	fbSetExtendedFadeTime.ipDALICommunication := ipDALICommunication;
	fbSetFadeRate.ipDALICommunication := ipDALICommunication;
	fbSetFadeTime.ipDALICommunication := ipDALICommunication;
{endregion}
10:
{region "Query Fade Time and Fade Rate"}
	fbQueryFadeTimeFadeRate(bStart := TRUE,
							nAddress := nAddress,
							eAddressType := eAddressType,
							eCommandPriority := E_DALICommandPriority.Middle,
							eFadeTime=> eFadeTime,
							eFadeRate=> eFadeRate);
	IF (NOT fbQueryFadeTimeFadeRate.bBusy) THEN
		fbQueryFadeTimeFadeRate(bStart := FALSE);
		IF (eFadeTime = 0) THEN 
			bNoFadeTime := FALSE; // Check whether Fade Time is available
			nStep := 20;
		ELSE 	 
			bNoFadeTime := TRUE;
			nStep := 0;
		END_IF
	END_IF
{endregion}
20:
{region "Query Extended Fade Time"}
	fbQueryExtendedFadeTime(bStart := TRUE,
							nAddress := nAddress,
							eAddressType := eAddressType,
							eCommandPriority := E_DALICommandPriority.Middle,
							eExtendedFadeTimeBase=> eExtendedFadeTimeBase,
							eExtendedFadeTimeMultiplier=> eExtendedFadeTimeMultiplier);
	IF (NOT fbQueryExtendedFadeTime.bBusy) THEN
		fbQueryExtendedFadeTime(bStart := FALSE);
		nStep := 0;
		IF (eExtendedFadeTimeMultiplier = E_DALIExtendedFadeTimeMultiplier.Disabled) THEN
			eExtendedFadeTime := E_DALIExtendedFadeTime.NoFade;
		END_IF
		IF (eExtendedFadeTimeMultiplier = E_DALIExtendedFadeTimeMultiplier.Multiplier100ms) THEN
			CASE eExtendedFadeTimeBase OF
				E_DALIExtendedFadeTimeBase.Base01:	eExtendedFadeTime := E_DALIExtendedFadeTime.onehundred;
				E_DALIExtendedFadeTimeBase.Base02:	eExtendedFadeTime := E_DALIExtendedFadeTime.twohundred;
				E_DALIExtendedFadeTimeBase.Base03:	eExtendedFadeTime := E_DALIExtendedFadeTime.threehundred;
				E_DALIExtendedFadeTimeBase.Base04:	eExtendedFadeTime := E_DALIExtendedFadeTime.fourhundred;
				E_DALIExtendedFadeTimeBase.Base05:	eExtendedFadeTime := E_DALIExtendedFadeTime.fivehundred;
				E_DALIExtendedFadeTimeBase.Base06:	eExtendedFadeTime := E_DALIExtendedFadeTime.sixhundred;
				E_DALIExtendedFadeTimeBase.Base07:	eExtendedFadeTime := E_DALIExtendedFadeTime.sevenhundred;
				E_DALIExtendedFadeTimeBase.Base08:	eExtendedFadeTime := E_DALIExtendedFadeTime.eighthundred;
				E_DALIExtendedFadeTimeBase.Base09:	eExtendedFadeTime := E_DALIExtendedFadeTime.ninehundred;
				E_DALIExtendedFadeTimeBase.Base10:	eExtendedFadeTime := E_DALIExtendedFadeTime.onethousand;
				E_DALIExtendedFadeTimeBase.Base11:	eExtendedFadeTime := E_DALIExtendedFadeTime.onethousandonehundred;
				E_DALIExtendedFadeTimeBase.Base12:	eExtendedFadeTime := E_DALIExtendedFadeTime.onethousandtwohundred;
				E_DALIExtendedFadeTimeBase.Base13:	eExtendedFadeTime := E_DALIExtendedFadeTime.onethousandthreehundred;
				E_DALIExtendedFadeTimeBase.Base14:	eExtendedFadeTime := E_DALIExtendedFadeTime.onethousandfourhundred;
				E_DALIExtendedFadeTimeBase.Base15:	eExtendedFadeTime := E_DALIExtendedFadeTime.onethousandfivehundred;
				E_DALIExtendedFadeTimeBase.Base16:	eExtendedFadeTime := E_DALIExtendedFadeTime.onethousandsixhundred;
			END_CASE
		END_IF
	 	IF (eExtendedFadeTimeMultiplier = E_DALIExtendedFadeTimeMultiplier.Multiplier1s) THEN
			CASE eExtendedFadeTimeBase OF
				E_DALIExtendedFadeTimeBase.Base01:	eExtendedFadeTime := E_DALIExtendedFadeTime.onesecond;
				E_DALIExtendedFadeTimeBase.Base02:	eExtendedFadeTime := E_DALIExtendedFadeTime.twoseconds;
				E_DALIExtendedFadeTimeBase.Base03:	eExtendedFadeTime := E_DALIExtendedFadeTime.threeseconds;
				E_DALIExtendedFadeTimeBase.Base04:	eExtendedFadeTime := E_DALIExtendedFadeTime.fourseconds;
				E_DALIExtendedFadeTimeBase.Base05:	eExtendedFadeTime := E_DALIExtendedFadeTime.fiveseconds;
				E_DALIExtendedFadeTimeBase.Base06:	eExtendedFadeTime := E_DALIExtendedFadeTime.sixseconds;
				E_DALIExtendedFadeTimeBase.Base07:	eExtendedFadeTime := E_DALIExtendedFadeTime.sevenseconds;
				E_DALIExtendedFadeTimeBase.Base08:	eExtendedFadeTime := E_DALIExtendedFadeTime.eightseconds;
				E_DALIExtendedFadeTimeBase.Base09:	eExtendedFadeTime := E_DALIExtendedFadeTime.nineseconds;
				E_DALIExtendedFadeTimeBase.Base10:	eExtendedFadeTime := E_DALIExtendedFadeTime.tenseconds;
				E_DALIExtendedFadeTimeBase.Base11:	eExtendedFadeTime := E_DALIExtendedFadeTime.elevenseconds;
				E_DALIExtendedFadeTimeBase.Base12:	eExtendedFadeTime := E_DALIExtendedFadeTime.twelveseconds;
				E_DALIExtendedFadeTimeBase.Base13:	eExtendedFadeTime := E_DALIExtendedFadeTime.thirteenseconds;
				E_DALIExtendedFadeTimeBase.Base14:	eExtendedFadeTime := E_DALIExtendedFadeTime.fourteenseconds;
				E_DALIExtendedFadeTimeBase.Base15:	eExtendedFadeTime := E_DALIExtendedFadeTime.fifteenseconds;
				E_DALIExtendedFadeTimeBase.Base16:	eExtendedFadeTime := E_DALIExtendedFadeTime.sixteenseconds;
			END_CASE
		END_IF
		IF (eExtendedFadeTimeMultiplier = E_DALIExtendedFadeTimeMultiplier.Multiplier10s) THEN
			CASE eExtendedFadeTimeBase OF
				E_DALIExtendedFadeTimeBase.Base01:	eExtendedFadeTime := E_DALIExtendedFadeTime.ten1seconds;
				E_DALIExtendedFadeTimeBase.Base02:	eExtendedFadeTime := E_DALIExtendedFadeTime.twentyseconds;
				E_DALIExtendedFadeTimeBase.Base03:	eExtendedFadeTime := E_DALIExtendedFadeTime.thirtyseconds;
				E_DALIExtendedFadeTimeBase.Base04:	eExtendedFadeTime := E_DALIExtendedFadeTime.fourtyseconds;
				E_DALIExtendedFadeTimeBase.Base05:	eExtendedFadeTime := E_DALIExtendedFadeTime.fiftyseconds;
				E_DALIExtendedFadeTimeBase.Base06:	eExtendedFadeTime := E_DALIExtendedFadeTime.sixtyseconds;
				E_DALIExtendedFadeTimeBase.Base07:	eExtendedFadeTime := E_DALIExtendedFadeTime.seventyseconds;
				E_DALIExtendedFadeTimeBase.Base08:	eExtendedFadeTime := E_DALIExtendedFadeTime.eightyseconds;
				E_DALIExtendedFadeTimeBase.Base09:	eExtendedFadeTime := E_DALIExtendedFadeTime.ninetyseconds;
				E_DALIExtendedFadeTimeBase.Base10:	eExtendedFadeTime := E_DALIExtendedFadeTime.onehundredseconds;
				E_DALIExtendedFadeTimeBase.Base11:	eExtendedFadeTime := E_DALIExtendedFadeTime.onehundredtenseconds;
				E_DALIExtendedFadeTimeBase.Base12:	eExtendedFadeTime := E_DALIExtendedFadeTime.onehundredtwentyseconds;
				E_DALIExtendedFadeTimeBase.Base13:	eExtendedFadeTime := E_DALIExtendedFadeTime.onehundredthirtyseconds;
				E_DALIExtendedFadeTimeBase.Base14:	eExtendedFadeTime := E_DALIExtendedFadeTime.onehundredfourtyseconds;
				E_DALIExtendedFadeTimeBase.Base15:	eExtendedFadeTime := E_DALIExtendedFadeTime.onehundredfiftyseconds;
				E_DALIExtendedFadeTimeBase.Base16:	eExtendedFadeTime := E_DALIExtendedFadeTime.onehundredsixtyseconds;
			END_CASE
		END_IF
		IF (eExtendedFadeTimeMultiplier = E_DALIExtendedFadeTimeMultiplier.Multiplier1min) THEN
			CASE eExtendedFadeTimeBase OF
				E_DALIExtendedFadeTimeBase.Base01:	eExtendedFadeTime := E_DALIExtendedFadeTime.oneminute;
				E_DALIExtendedFadeTimeBase.Base02:	eExtendedFadeTime := E_DALIExtendedFadeTime.twominutes;
				E_DALIExtendedFadeTimeBase.Base03:	eExtendedFadeTime := E_DALIExtendedFadeTime.threeminutes;
				E_DALIExtendedFadeTimeBase.Base04:	eExtendedFadeTime := E_DALIExtendedFadeTime.fourminutes;
				E_DALIExtendedFadeTimeBase.Base05:	eExtendedFadeTime := E_DALIExtendedFadeTime.fiveminutes;
				E_DALIExtendedFadeTimeBase.Base06:	eExtendedFadeTime := E_DALIExtendedFadeTime.sixminutes;
				E_DALIExtendedFadeTimeBase.Base07:	eExtendedFadeTime := E_DALIExtendedFadeTime.sevenminutes;
				E_DALIExtendedFadeTimeBase.Base08:	eExtendedFadeTime := E_DALIExtendedFadeTime.eightminutes;
				E_DALIExtendedFadeTimeBase.Base09:	eExtendedFadeTime := E_DALIExtendedFadeTime.nineminutes;
				E_DALIExtendedFadeTimeBase.Base10:	eExtendedFadeTime := E_DALIExtendedFadeTime.tenminutes;
				E_DALIExtendedFadeTimeBase.Base11:	eExtendedFadeTime := E_DALIExtendedFadeTime.elevenminutes;
				E_DALIExtendedFadeTimeBase.Base12:	eExtendedFadeTime := E_DALIExtendedFadeTime.twelveminutes;
				E_DALIExtendedFadeTimeBase.Base13:	eExtendedFadeTime := E_DALIExtendedFadeTime.thirteenminutes;
				E_DALIExtendedFadeTimeBase.Base14:	eExtendedFadeTime := E_DALIExtendedFadeTime.fourteenminutes;
				E_DALIExtendedFadeTimeBase.Base15:	eExtendedFadeTime := E_DALIExtendedFadeTime.fifteenminutes;
				E_DALIExtendedFadeTimeBase.Base16:	eExtendedFadeTime := E_DALIExtendedFadeTime.sixteenminutes;
			END_CASE
		END_IF
	ELSE
		eExtendedFadeTime := E_DALIExtendedFadeTime.unknown;
	END_IF
{endregion}
1000:
{region "Set Fade Time"}
	fbSetFadeTime(bStart:= TRUE,
				  nAddress:= nAddress,
				  eAddressType := eAddressType,
				  eCommandPriority := E_DALICommandPriority.Middle,
				  eFadeTime := eFadeTime);
	IF (NOT fbSetFadeTime.bBusy) THEN
		fbSetFadeTime(bStart := FALSE);
		{region " Display whether Fade Time is available²}
		IF (eFadeTime = 0) THEN
			bNoFadeTime := FALSE;
		ELSE
			bNoFadeTime := TRUE;
		END_IF
		{endregion}
		nStep := 0;
	END_IF
{endregion}
1010:
{region "Set Fade Rate"}
	fbSetFadeRate(bStart:= TRUE,
				  nAddress:= nAddress,
				  eAddressType := eAddressType,
				  eCommandPriority := E_DALICommandPriority.Middle,
				  eFadeRate := eFadeRate);
	IF (NOT fbSetFadeRate.bBusy) THEN
		fbSetFadeRate(bStart := FALSE);
		nStep := 0;
	END_IF
{endregion}
1020:
{region "Set Extended Fade Time"}
	CASE eExtendedFadeTime OF
		E_DALIExtendedFadeTime.NoFade:					eExtendedFadeTimeBase := E_DALIExtendedFadeTimeBase.Unknown;
														eExtendedFadeTimeMultiplier := E_DALIExtendedFadeTimeMultiplier.Disabled;
		E_DALIExtendedFadeTime.onehundred:				eExtendedFadeTimeBase := E_DALIExtendedFadeTimeBase.Base01;
														eExtendedFadeTimeMultiplier := E_DALIExtendedFadeTimeMultiplier.Multiplier100ms;
		E_DALIExtendedFadeTime.twohundred:				eExtendedFadeTimeBase := E_DALIExtendedFadeTimeBase.Base02;
														eExtendedFadeTimeMultiplier := E_DALIExtendedFadeTimeMultiplier.Multiplier100ms;
		E_DALIExtendedFadeTime.threehundred:			eExtendedFadeTimeBase := E_DALIExtendedFadeTimeBase.Base03;
														eExtendedFadeTimeMultiplier := E_DALIExtendedFadeTimeMultiplier.Multiplier100ms;
		E_DALIExtendedFadeTime.fourhundred:				eExtendedFadeTimeBase := E_DALIExtendedFadeTimeBase.Base04;
														eExtendedFadeTimeMultiplier := E_DALIExtendedFadeTimeMultiplier.Multiplier100ms;
		E_DALIExtendedFadeTime.fivehundred:				eExtendedFadeTimeBase := E_DALIExtendedFadeTimeBase.Base05;
														eExtendedFadeTimeMultiplier := E_DALIExtendedFadeTimeMultiplier.Multiplier100ms;
		E_DALIExtendedFadeTime.sixhundred:				eExtendedFadeTimeBase := E_DALIExtendedFadeTimeBase.Base06;
														eExtendedFadeTimeMultiplier := E_DALIExtendedFadeTimeMultiplier.Multiplier100ms;
		E_DALIExtendedFadeTime.sevenhundred:			eExtendedFadeTimeBase := E_DALIExtendedFadeTimeBase.Base07;
														eExtendedFadeTimeMultiplier := E_DALIExtendedFadeTimeMultiplier.Multiplier100ms;
		E_DALIExtendedFadeTime.eighthundred:			eExtendedFadeTimeBase := E_DALIExtendedFadeTimeBase.Base08;
														eExtendedFadeTimeMultiplier := E_DALIExtendedFadeTimeMultiplier.Multiplier100ms;
		E_DALIExtendedFadeTime.ninehundred:				eExtendedFadeTimeBase := E_DALIExtendedFadeTimeBase.Base09;
														eExtendedFadeTimeMultiplier := E_DALIExtendedFadeTimeMultiplier.Multiplier100ms;
		E_DALIExtendedFadeTime.onethousand:				eExtendedFadeTimeBase := E_DALIExtendedFadeTimeBase.Base10;
														eExtendedFadeTimeMultiplier := E_DALIExtendedFadeTimeMultiplier.Multiplier100ms;
		E_DALIExtendedFadeTime.onethousandonehundred:	eExtendedFadeTimeBase := E_DALIExtendedFadeTimeBase.Base11;
														eExtendedFadeTimeMultiplier := E_DALIExtendedFadeTimeMultiplier.Multiplier100ms;
		E_DALIExtendedFadeTime.onethousandtwohundred:	eExtendedFadeTimeBase := E_DALIExtendedFadeTimeBase.Base12;
														eExtendedFadeTimeMultiplier := E_DALIExtendedFadeTimeMultiplier.Multiplier100ms;
		E_DALIExtendedFadeTime.onethousandthreehundred:	eExtendedFadeTimeBase := E_DALIExtendedFadeTimeBase.Base13;
														eExtendedFadeTimeMultiplier := E_DALIExtendedFadeTimeMultiplier.Multiplier100ms;
		E_DALIExtendedFadeTime.onethousandfourhundred:	eExtendedFadeTimeBase := E_DALIExtendedFadeTimeBase.Base14;
														eExtendedFadeTimeMultiplier := E_DALIExtendedFadeTimeMultiplier.Multiplier100ms;
		E_DALIExtendedFadeTime.onethousandfivehundred:	eExtendedFadeTimeBase := E_DALIExtendedFadeTimeBase.Base15;
														eExtendedFadeTimeMultiplier := E_DALIExtendedFadeTimeMultiplier.Multiplier100ms;
		E_DALIExtendedFadeTime.onethousandsixhundred:	eExtendedFadeTimeBase := E_DALIExtendedFadeTimeBase.Base16;
														eExtendedFadeTimeMultiplier := E_DALIExtendedFadeTimeMultiplier.Multiplier100ms;
		E_DALIExtendedFadeTime.onesecond:				eExtendedFadeTimeBase := E_DALIExtendedFadeTimeBase.Base01;
														eExtendedFadeTimeMultiplier := E_DALIExtendedFadeTimeMultiplier.Multiplier1s;
		E_DALIExtendedFadeTime.twoseconds:				eExtendedFadeTimeBase := E_DALIExtendedFadeTimeBase.Base02;
														eExtendedFadeTimeMultiplier := E_DALIExtendedFadeTimeMultiplier.Multiplier1s;
		E_DALIExtendedFadeTime.threeseconds:			eExtendedFadeTimeBase := E_DALIExtendedFadeTimeBase.Base03;
														eExtendedFadeTimeMultiplier := E_DALIExtendedFadeTimeMultiplier.Multiplier1s;
		E_DALIExtendedFadeTime.fourseconds:				eExtendedFadeTimeBase := E_DALIExtendedFadeTimeBase.Base04;
														eExtendedFadeTimeMultiplier := E_DALIExtendedFadeTimeMultiplier.Multiplier1s;
		E_DALIExtendedFadeTime.fiveseconds:				eExtendedFadeTimeBase := E_DALIExtendedFadeTimeBase.Base05;
														eExtendedFadeTimeMultiplier := E_DALIExtendedFadeTimeMultiplier.Multiplier1s;
		E_DALIExtendedFadeTime.sixseconds:				eExtendedFadeTimeBase := E_DALIExtendedFadeTimeBase.Base06;
														eExtendedFadeTimeMultiplier := E_DALIExtendedFadeTimeMultiplier.Multiplier1s;
		E_DALIExtendedFadeTime.sevenseconds:			eExtendedFadeTimeBase := E_DALIExtendedFadeTimeBase.Base07;
														eExtendedFadeTimeMultiplier := E_DALIExtendedFadeTimeMultiplier.Multiplier1s;
		E_DALIExtendedFadeTime.eightseconds:			eExtendedFadeTimeBase := E_DALIExtendedFadeTimeBase.Base08;
														eExtendedFadeTimeMultiplier := E_DALIExtendedFadeTimeMultiplier.Multiplier1s;
		E_DALIExtendedFadeTime.nineseconds:				eExtendedFadeTimeBase := E_DALIExtendedFadeTimeBase.Base09;
														eExtendedFadeTimeMultiplier := E_DALIExtendedFadeTimeMultiplier.Multiplier1s;
		E_DALIExtendedFadeTime.tenseconds:				eExtendedFadeTimeBase := E_DALIExtendedFadeTimeBase.Base10;
														eExtendedFadeTimeMultiplier := E_DALIExtendedFadeTimeMultiplier.Multiplier1s;
		E_DALIExtendedFadeTime.elevenseconds:			eExtendedFadeTimeBase := E_DALIExtendedFadeTimeBase.Base11;
														eExtendedFadeTimeMultiplier := E_DALIExtendedFadeTimeMultiplier.Multiplier1s;
		E_DALIExtendedFadeTime.twelveseconds:			eExtendedFadeTimeBase := E_DALIExtendedFadeTimeBase.Base12;
														eExtendedFadeTimeMultiplier := E_DALIExtendedFadeTimeMultiplier.Multiplier1s;
		E_DALIExtendedFadeTime.thirteenseconds:			eExtendedFadeTimeBase := E_DALIExtendedFadeTimeBase.Base13;
														eExtendedFadeTimeMultiplier := E_DALIExtendedFadeTimeMultiplier.Multiplier1s;
		E_DALIExtendedFadeTime.fourteenseconds:			eExtendedFadeTimeBase := E_DALIExtendedFadeTimeBase.Base14;
														eExtendedFadeTimeMultiplier := E_DALIExtendedFadeTimeMultiplier.Multiplier1s;
		E_DALIExtendedFadeTime.fifteenseconds:			eExtendedFadeTimeBase := E_DALIExtendedFadeTimeBase.Base15;
														eExtendedFadeTimeMultiplier := E_DALIExtendedFadeTimeMultiplier.Multiplier1s;
		E_DALIExtendedFadeTime.sixteenseconds:			eExtendedFadeTimeBase := E_DALIExtendedFadeTimeBase.Base16;
														eExtendedFadeTimeMultiplier := E_DALIExtendedFadeTimeMultiplier.Multiplier1s;
		E_DALIExtendedFadeTime.ten1seconds:				eExtendedFadeTimeBase := E_DALIExtendedFadeTimeBase.Base01;
														eExtendedFadeTimeMultiplier := E_DALIExtendedFadeTimeMultiplier.Multiplier10s;
		E_DALIExtendedFadeTime.twentyseconds:			eExtendedFadeTimeBase := E_DALIExtendedFadeTimeBase.Base02;
														eExtendedFadeTimeMultiplier := E_DALIExtendedFadeTimeMultiplier.Multiplier10s;
		E_DALIExtendedFadeTime.thirtyseconds:			eExtendedFadeTimeBase := E_DALIExtendedFadeTimeBase.Base03;
														eExtendedFadeTimeMultiplier := E_DALIExtendedFadeTimeMultiplier.Multiplier10s;
		E_DALIExtendedFadeTime.fourtyseconds:			eExtendedFadeTimeBase := E_DALIExtendedFadeTimeBase.Base04;
														eExtendedFadeTimeMultiplier := E_DALIExtendedFadeTimeMultiplier.Multiplier10s;
		E_DALIExtendedFadeTime.fiftyseconds:			eExtendedFadeTimeBase := E_DALIExtendedFadeTimeBase.Base05;
														eExtendedFadeTimeMultiplier := E_DALIExtendedFadeTimeMultiplier.Multiplier10s;
		E_DALIExtendedFadeTime.sixtyseconds:			eExtendedFadeTimeBase := E_DALIExtendedFadeTimeBase.Base06;
														eExtendedFadeTimeMultiplier := E_DALIExtendedFadeTimeMultiplier.Multiplier10s;
		E_DALIExtendedFadeTime.seventyseconds:			eExtendedFadeTimeBase := E_DALIExtendedFadeTimeBase.Base07;
														eExtendedFadeTimeMultiplier := E_DALIExtendedFadeTimeMultiplier.Multiplier10s;
		E_DALIExtendedFadeTime.eightyseconds:			eExtendedFadeTimeBase := E_DALIExtendedFadeTimeBase.Base08;
														eExtendedFadeTimeMultiplier := E_DALIExtendedFadeTimeMultiplier.Multiplier10s;
		E_DALIExtendedFadeTime.ninetyseconds:			eExtendedFadeTimeBase := E_DALIExtendedFadeTimeBase.Base09;
														eExtendedFadeTimeMultiplier := E_DALIExtendedFadeTimeMultiplier.Multiplier10s;
		E_DALIExtendedFadeTime.onehundredseconds:		eExtendedFadeTimeBase := E_DALIExtendedFadeTimeBase.Base10;
														eExtendedFadeTimeMultiplier := E_DALIExtendedFadeTimeMultiplier.Multiplier10s;
		E_DALIExtendedFadeTime.onehundredtenseconds:	eExtendedFadeTimeBase := E_DALIExtendedFadeTimeBase.Base11;
														eExtendedFadeTimeMultiplier := E_DALIExtendedFadeTimeMultiplier.Multiplier10s;
		E_DALIExtendedFadeTime.onehundredtwentyseconds:	eExtendedFadeTimeBase := E_DALIExtendedFadeTimeBase.Base12;
														eExtendedFadeTimeMultiplier := E_DALIExtendedFadeTimeMultiplier.Multiplier10s;
		E_DALIExtendedFadeTime.onehundredthirtyseconds:	eExtendedFadeTimeBase := E_DALIExtendedFadeTimeBase.Base13;
														eExtendedFadeTimeMultiplier := E_DALIExtendedFadeTimeMultiplier.Multiplier10s;
		E_DALIExtendedFadeTime.onehundredfourtyseconds:	eExtendedFadeTimeBase := E_DALIExtendedFadeTimeBase.Base14;
														eExtendedFadeTimeMultiplier := E_DALIExtendedFadeTimeMultiplier.Multiplier10s;
		E_DALIExtendedFadeTime.onehundredfiftyseconds:	eExtendedFadeTimeBase := E_DALIExtendedFadeTimeBase.Base15;
														eExtendedFadeTimeMultiplier := E_DALIExtendedFadeTimeMultiplier.Multiplier10s;
		E_DALIExtendedFadeTime.onehundredsixtyseconds:	eExtendedFadeTimeBase := E_DALIExtendedFadeTimeBase.Base16;
														eExtendedFadeTimeMultiplier := E_DALIExtendedFadeTimeMultiplier.Multiplier10s;
		E_DALIExtendedFadeTime.oneminute:				eExtendedFadeTimeBase := E_DALIExtendedFadeTimeBase.Base01;
														eExtendedFadeTimeMultiplier := E_DALIExtendedFadeTimeMultiplier.Multiplier1min;
		E_DALIExtendedFadeTime.twominutes:				eExtendedFadeTimeBase := E_DALIExtendedFadeTimeBase.Base02;
														eExtendedFadeTimeMultiplier := E_DALIExtendedFadeTimeMultiplier.Multiplier1min;
		E_DALIExtendedFadeTime.threeminutes:			eExtendedFadeTimeBase := E_DALIExtendedFadeTimeBase.Base03;
														eExtendedFadeTimeMultiplier := E_DALIExtendedFadeTimeMultiplier.Multiplier1min;
		E_DALIExtendedFadeTime.fourminutes:				eExtendedFadeTimeBase := E_DALIExtendedFadeTimeBase.Base04;
														eExtendedFadeTimeMultiplier := E_DALIExtendedFadeTimeMultiplier.Multiplier1min;
		E_DALIExtendedFadeTime.fiveminutes:				eExtendedFadeTimeBase := E_DALIExtendedFadeTimeBase.Base05;
														eExtendedFadeTimeMultiplier := E_DALIExtendedFadeTimeMultiplier.Multiplier1min;
		E_DALIExtendedFadeTime.sixminutes:				eExtendedFadeTimeBase := E_DALIExtendedFadeTimeBase.Base06;
														eExtendedFadeTimeMultiplier := E_DALIExtendedFadeTimeMultiplier.Multiplier1min;
		E_DALIExtendedFadeTime.sevenminutes:			eExtendedFadeTimeBase := E_DALIExtendedFadeTimeBase.Base07;
														eExtendedFadeTimeMultiplier := E_DALIExtendedFadeTimeMultiplier.Multiplier1min;
		E_DALIExtendedFadeTime.eightminutes:			eExtendedFadeTimeBase := E_DALIExtendedFadeTimeBase.Base08;
														eExtendedFadeTimeMultiplier := E_DALIExtendedFadeTimeMultiplier.Multiplier1min;
		E_DALIExtendedFadeTime.nineminutes:				eExtendedFadeTimeBase := E_DALIExtendedFadeTimeBase.Base09;
														eExtendedFadeTimeMultiplier := E_DALIExtendedFadeTimeMultiplier.Multiplier1min;
		E_DALIExtendedFadeTime.tenminutes:				eExtendedFadeTimeBase := E_DALIExtendedFadeTimeBase.Base10;
														eExtendedFadeTimeMultiplier := E_DALIExtendedFadeTimeMultiplier.Multiplier1min;
		E_DALIExtendedFadeTime.elevenminutes:			eExtendedFadeTimeBase := E_DALIExtendedFadeTimeBase.Base11;
														eExtendedFadeTimeMultiplier := E_DALIExtendedFadeTimeMultiplier.Multiplier1min;
		E_DALIExtendedFadeTime.twelveminutes:			eExtendedFadeTimeBase := E_DALIExtendedFadeTimeBase.Base12;
														eExtendedFadeTimeMultiplier := E_DALIExtendedFadeTimeMultiplier.Multiplier1min;
		E_DALIExtendedFadeTime.thirteenminutes:			eExtendedFadeTimeBase := E_DALIExtendedFadeTimeBase.Base13;
														eExtendedFadeTimeMultiplier := E_DALIExtendedFadeTimeMultiplier.Multiplier1min;
		E_DALIExtendedFadeTime.fourteenminutes:			eExtendedFadeTimeBase := E_DALIExtendedFadeTimeBase.Base14;
														eExtendedFadeTimeMultiplier := E_DALIExtendedFadeTimeMultiplier.Multiplier1min;
		E_DALIExtendedFadeTime.fifteenminutes:			eExtendedFadeTimeBase := E_DALIExtendedFadeTimeBase.Base15;
														eExtendedFadeTimeMultiplier := E_DALIExtendedFadeTimeMultiplier.Multiplier1min;
		E_DALIExtendedFadeTime.sixteenminutes:			eExtendedFadeTimeBase := E_DALIExtendedFadeTimeBase.Base16;
														eExtendedFadeTimeMultiplier := E_DALIExtendedFadeTimeMultiplier.Multiplier1min;
		E_DALIExtendedFadeTime.unknown:					eExtendedFadeTimeBase := E_DALIExtendedFadeTimeBase.Unknown;
														eExtendedFadeTimeMultiplier := E_DALIExtendedFadeTimeMultiplier.Unknown;
	END_CASE
	fbSetExtendedFadeTime(bStart:= TRUE,
						  nAddress:= nAddress,
						  eAddressType := eAddressType,
						  eCommandPriority := E_DALICommandPriority.Middle,
						  eExtendedFadeTimeBase := eExtendedFadeTimeBase,
						  eExtendedFadeTimeMultiplier := eExtendedFadeTimeMultiplier);
	IF (NOT fbSetExtendedFadeTime.bBusy) THEN
		fbSetExtendedFadeTime(bStart := FALSE);
		nStep := 0;
	END_IF
{endregion}
END_CASE

END_FUNCTION_BLOCK

// ---- GlobalTextList.TcGTLO
TEXTLIST GlobalTextList
  621 = '%d'
  665 = '%d %'
  2025 = '%d ms'
  1540 = '%d s'
  646 = '%s'
  640 = '0'
  641 = '1'
  661 = '10'
  662 = '11'
  663 = '12'
  999 = '13'
  1000 = '14'
  1001 = '15'
  1002 = '16'
  1003 = '17'
  1004 = '18'
  1005 = '19'
  642 = '2'
  1006 = '20'
  1007 = '21'
  1008 = '22'
  1009 = '23'
  1010 = '24'
  1011 = '25'
  1012 = '26'
  1013 = '27'
  1014 = '28'
  1015 = '29'
  654 = '3'
  1016 = '30'
  1017 = '31'
  1018 = '32'
  1019 = '33'
  1020 = '34'
  1021 = '35'
  1022 = '36'
  1023 = '37'
  1024 = '38'
  1025 = '39'
  655 = '4'
  1026 = '40'
  1027 = '41'
  1028 = '42'
  1029 = '43'
  1030 = '44'
  1031 = '45'
  1032 = '46'
  1033 = '47'
  1034 = '48'
  1035 = '49'
  656 = '5'
  358 = '50'
  359 = '51'
  360 = '52'
  361 = '53'
  362 = '54'
  363 = '55'
  364 = '56'
  365 = '57'
  366 = '58'
  367 = '59'
  657 = '6'
  368 = '60'
  369 = '61'
  370 = '62'
  371 = '63'
  658 = '7'
  659 = '8'
  660 = '9'
  1089 = 'AC-supply possible'
  644 = 'Actual Level:'
  650 = 'Address Type'
  1175 = 'AM Operation active:'
  1044 = 'AM operation possible'
  2131 = 'Back'
  2471 = 'Bit 0'
  379 = 'Bit 1'
  2734 = 'Bit 2'
  2320 = 'Bit 3'
  929 = 'Bit 4'
  2576 = 'Bit 5'
  2065 = 'Bit 6'
  1623 = 'Bit 7'
  803 = 'Broadcast'
  515 = 'Button pressed'
  498 = 'Button released'
  527 = 'Button stuck / free'
  593 = 'Cancel Hold Timer'
  2101 = 'Catch Movement'
  2319 = 'Catching:'
  897 = 'Change Addresses'
  372 = 'Choose group:'
  98 = 'Choose scene:'
  618 = 'Complete new installation \n(all addresses will be removed)'
  807 = 'Control'
  645 = 'Control Gear Failure:'
  146 = 'Control LED'
  445 = 'Current protection active:'
  1716 = 'Current protection device'
  668 = 'Current protection enabled:'
  5 = 'Current Protector Enabled '
  1902 = 'DALI Line:'
  334 = 'DALI Power Supply'
  1135 = 'DC-supply possible'
  560 = 'Deadtime Timer:'
  1180 = 'DI1 falling edge'
  1218 = 'DI1 rising edge'
  1726 = 'DI2 falling edge'
  1876 = 'DI2 rising edge'
  936 = 'Dimming Curve:'
  169 = 'Do not lock process image'
  2135 = 'Do not lock process image in case of \nDALI commands from DI1 or DI2'
  2344 = 'Do not lock process image in case of DALI commands from DI1 or DI2'
  519 = 'Double press'
  1112 = 'Double Timer Min:'
  482 = 'Double Timer:'
  811 = 'Down'
  486 = 'Enable'
  828 = 'Enable:'
  1982 = 'EventPriority'
  32 = 'EventPriority:'
  494 = 'EventScheme'
  1113 = 'EventScheme:'
  1841 = 'Extended Fade Time only valid if Fade Time equals 0!'
  310 = 'Extended Version Number'
  649 = 'Fade Running:'
  1150 = 'FadeRate'
  1160 = 'FadeTime'
  319 = 'Fast Fade Time:'
  1808 = 'Features LED'
  1434 = 'GearType LED'
  815 = 'Go to Scene'
  99 = 'Go to scene'
  802 = 'Group Address'
  1923 = 'Hier noch die Abfrage der extended version Number\nmit reinbringen, damit klar wird welcher Edition das Gerät angehört.'
  568 = 'Hold Timer:'
  311 = 'Hysteresis Min:'
  313 = 'Hysteresis:'
  1117 = 'Identify'
  2159 = 'Identify 202'
  315 = 'Illuminance Level'
  540 = 'Input Value:'
  544 = 'Instance Error:'
  1038 = 'Instance Number:'
  1374 = 'InstanceType0'
  652 = 'InstanceType1'
  653 = 'InstanceType3'
  664 = 'InstanceType4'
  492 = 'Internal DALI power supply disabled'
  1820 = 'IT0 (Generic Input)'
  1151 = 'IT1 (PushButton)'
  906 = 'IT2 (absolute Input)'
  909 = 'IT2 (Absolute Input)'
  819 = 'IT3 (Occupancy)'
  224 = 'IT4 (Light Sensor)'
  1771 = 'K-Bus Watchdog'
  647 = 'Lamp Failure:'
  506 = 'LED module integrated'
  306 = 'Load Decrease:'
  1137 = 'Load Increase:'
  1811 = 'Lockable bytes: changeable if "Offset 2" has the Value 85 (0x55).\nFor changing use decimal value.'
  523 = 'Long press repeat'
  507 = 'Long press start'
  511 = 'Long press stop'
  2046 = 'Memory Bank:'
  584 = 'Movement'
  531 = 'na'
  842 = 'Name'
  926 = 'Name of byte in memory bank'
  193 = 'NewAddress'
  588 = 'No Movement'
  572 = 'Occupied'
  808 = 'Off'
  835 = 'Offset'
  1329 = 'Offset in memory bank'
  192 = 'OldAddress'
  816 = 'On and Step Up'
  277 = 'Open Circuit:'
  651 = 'OperatingMode'
  619 = 'Optical feedback'
  963 = 'Output is current controlled'
  826 = 'Output regulated by current:'
  1900 = 'Parameters'
  2547 = 'Parameters Absolute Input Device'
  1580 = 'Parameters Generic Instance'
  309 = 'Parameters Light Sensor'
  556 = 'Parameters Occupancy Sensor'
  465 = 'Parameters Pushbutton Sensor'
  1847 = 'Physical selection supported'
  1071 = 'Please check if Current Protector is present \nby reading parameters first.'
  308 = 'Please select the desired Short Address in the table above.'
  751 = 'Position Event'
  930 = 'Possible Operating Modes LED'
  719 = 'Power pulse operation'
  1744 = 'Power supply integrated'
  1561 = 'PP Operation active:'
  970 = 'PWM Operation active:'
  1882 = 'PWM operation possible'
  1487 = 'Query idle time detection \nenabled'
  701 = 'Query load decrease enabled'
  1351 = 'Query load increase enabled'
  837 = 'Query reduction luminous flux \nregarding thermal overload'
  463 = 'Query short circuit enabled'
  1293 = 'Query thermal switch enabled'
  617 = 'Random Addressing'
  373 = 'Read'
  316 = 'Read parameters'
  181 = 'Read Parameters'
  1531 = 'Reads all Fading Parameters'
  810 = 'Recall Max Level'
  809 = 'Recall Min Level'
  186 = 'Ref. Measurement failed:'
  439 = 'Reference System Power'
  580 = 'Repeat'
  470 = 'Repeat Timer:'
  564 = 'Report Timer:'
  2418 = 'Reset inactive process image'
  648 = 'Reset State:'
  1037 = 'Resolution:'
  616 = 'Scan devices by address'
  1036 = 'Scene Level'
  814 = 'Scene:'
  1366 = 'Set Extended Fade Time'
  252 = 'Set Fade Rate'
  1875 = 'Set Fade Time'
  801 = 'Short Address'
  1179 = 'Short Address Range'
  1041 = 'Short Address:'
  34 = 'Short Circuit:'
  503 = 'Short press'
  1516 = 'Short Timer Min:'
  478 = 'Short Timer:'
  1170 = 'Single Short Address'
  615 = 'Start'
  620 = 'Start with address:'
  643 = 'Status'
  958 = 'Status Absolute Input Device'
  2506 = 'Status Generic Instance'
  82 = 'Status LED'
  317 = 'Status Light Sensor'
  597 = 'Status Occupancy Sensor'
  536 = 'Status Pushbutton Sensor'
  812 = 'Step Down'
  813 = 'Step Down and Off'
  818 = 'Step Up'
  164 = 'Stuck Timer:'
  376 = 'Switch Off'
  375 = 'Switch On'
  2458 = 'Terminal Event'
  1108 = 'Thermal Overload:'
  355 = 'Thermal Shut Down:'
  305 = 'To'
  804 = 'Unaddressed'
  817 = 'Up'
  2521 = 'V%s'
  298 = 'V3.1.1.0'
  858 = 'V3.4.0.0'
  395 = 'V3.4.0.1'
  1169 = 'V3.5.0.0'
  576 = 'Vacant'
  1205 = 'Value'
  850 = 'Value Dec'
  1435 = 'Value decimal'
  857 = 'Value Hex'
  2231 = 'Value hexadecimal,\nto change use\nvalue decimal'
  374 = 'Write'
  1047 = 'Write default values'
  490 = 'Write parameters'
END_TEXTLIST

// ---- VISUs/TextLists/DimmingCurve.TcTLO
TEXTLIST DimmingCurve
  0 = 'Logarithmic'
  1 = 'Linear'
  255 = 'Unknown'
   = ''
END_TEXTLIST

// ---- VISUs/TextLists/EventPriority.TcTLO
TEXTLIST EventPriority
  2 = 'MiddleHigh'
  3 = 'Middle'
  4 = 'MiddleLow'
  5 = 'Low'
  255 = 'Unknown'
   = ''
END_TEXTLIST

// ---- VISUs/TextLists/EventScheme.TcTLO
TEXTLIST EventScheme
  0 = '0 - Instance type and number'
  1 = '1 - Short address and instance type'
  2 = '2 - Short address and instance number'
  3 = '3 - Device group and instance type'
  4 = '4 - Instance group and instance type'
   = ''
END_TEXTLIST

// ---- VISUs/TextLists/ExtendedFadeTime.TcTLO
TEXTLIST ExtendedFadeTime
  0 = 'No Fade'
  1 = '1 * 100 ms = 100 ms'
  2 = '2 * 100 ms = 200 ms'
  3 = '3 * 100 ms = 300 ms'
  4 = '4 * 100 ms = 400 ms'
  5 = '5 * 100 ms = 500 ms'
  6 = '6 * 100 ms = 600 ms'
  7 = '7 * 100 ms = 700 ms'
  8 = '8 * 100 ms = 800 ms'
  9 = '9 * 100 ms = 900 ms'
  10 = '10 * 100 ms = 1000 ms'
  11 = '11 * 100 ms = 1100 ms'
  12 = '12 * 100 ms = 1200 ms'
  13 = '13 * 100 ms = 1300 ms'
  14 = '14 * 100 ms = 1400 ms'
  15 = '15 * 100 ms = 1500 ms'
  16 = '16 * 100 ms = 1600 ms'
  17 = '1 * 1 s = 1 s'
  18 = '2 * 1 s = 2 s'
  19 = '3 * 1 s = 3 s'
  20 = '4 * 1 s = 4 s'
  21 = '5 * 1 s = 5 s'
  22 = '6 * 1 s = 6 s'
  23 = '7 * 1 s = 7 s'
  24 = '8 * 1 s = 8 s'
  25 = '9 * 1 s = 9 s'
  26 = '10 * 1 s = 10 s'
  27 = '11 * 1 s = 11 s'
  28 = '12 * 1 s = 12 s'
  29 = '13 * 1 s = 13 s'
  30 = '14 * 1 s = 14 s'
  31 = '15 * 1 s = 15 s'
  32 = '16 * 1 s = 16 s'
  33 = '1 * 10 s = 10 s'
  34 = '2 * 10 s = 20 s'
  35 = '3 * 10 s = 30 s'
  36 = '4 * 10 s = 40 s'
  37 = '5 * 10 s = 50 s'
  38 = '6 * 10 s = 60 s'
  39 = '7 * 10 s = 70 s'
  40 = '8 * 10 s = 80 s'
  41 = '9 * 10 s = 90 s'
  42 = '10 * 10 s = 100 s'
  43 = '11 * 10 s = 110 s'
  44 = '12 * 10 s = 120 s'
  45 = '13 * 10 s = 130 s'
  46 = '14 * 10 s = 140 s'
  47 = '15 * 10 s = 150 s'
  48 = '16 * 10 s = 160 s'
  49 = '1 * 1 min = 1 min'
  50 = '2 * 1 min = 2 min'
  51 = '3 * 1 min = 3 min'
  52 = '4 * 1 min = 4 min'
  53 = '5 * 1 min = 5 min'
  54 = '6 * 1 min = 6 min'
  55 = '7 * 1 min = 7 min'
  56 = '8 * 1 min = 8 min'
  57 = '9 * 1 min = 9 min'
  58 = '10 * 1 min = 10 min'
  59 = '11 * 1 min = 11 min'
  60 = '12 * 1 min = 12 min'
  61 = '13 * 1 min = 13 min'
  62 = '14 * 1 min = 14 min'
  63 = '15 * 1 min = 15 min'
  64 = '16 * 1 min = 16 min'
  255 = 'Unknown'
   = ''
END_TEXTLIST

// ---- VISUs/TextLists/FadeRate.TcTLO
TEXTLIST FadeRate
  0 = 'Unknown'
  1 = '358 steps/s'
  2 = '253 steps/s'
  3 = '179 steps/s'
  4 = '127 steps/s'
  5 = '89,4 steps/s'
  6 = '63,3 steps/s'
  7 = '44,7 steps/s'
  8 = '31,6 steps/s'
  9 = '22,4 steps/s'
  10 = '15,8 steps/s'
  11 = '11,2 steps/s'
  12 = '7,9 steps/s'
  13 = '5,6 steps/s'
  14 = '4,0 steps/s'
  15 = '2,8 steps/s'
  255 = 'Unknown'
   = ''
END_TEXTLIST

// ---- VISUs/TextLists/FastFadeTime.TcTLO
TEXTLIST FastFadeTime
  0 = 'Disabled'
  4 = 'T100ms'
  8 = 'T200ms'
  12 = 'T300ms'
  16 = 'T400ms'
  20 = 'T500ms'
  24 = 'T600ms'
  27 = 'T700ms'
  255 = 'Unknown'
   = ''
END_TEXTLIST

// ---- VISUs/Visu_DALICommissioning/Visu_KL6821Configuration.TcVIS
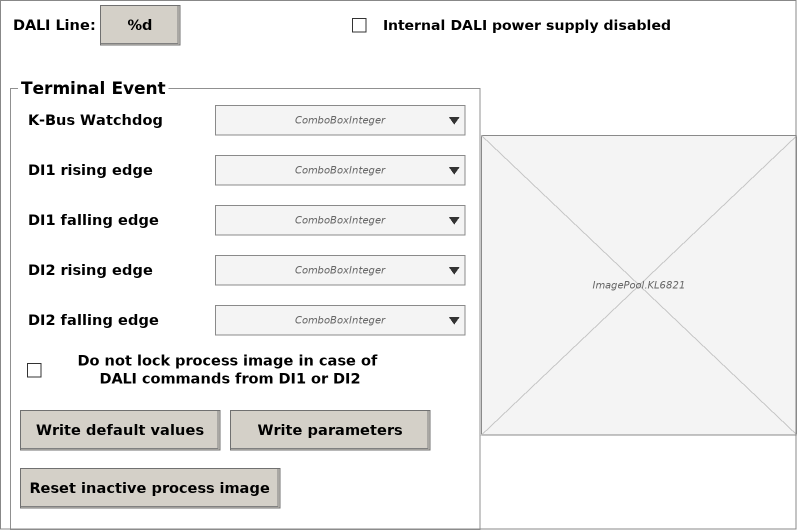
VISUALIZATION Visu_KL6821Configuration  // 797x530
    GroupBox (10,80 470x450), "Terminal Event"
        Textfield (15,25 170x30), "K-Bus Watchdog"
        ComboBoxInteger (205,25 250x30), variable: Communication.eCommandKBusWatchdog, text list: 'CommandOnTerminalEvent'
        Textfield (15,75 170x30), "DI1 rising edge"
        Textfield (15,125 170x30), "DI1 falling edge"
        ComboBoxInteger (205,75 250x30), variable: Communication.eCommandDI1RisingEdge, text list: 'CommandOnTerminalEvent'
        ComboBoxInteger (205,125 250x30), variable: Communication.eCommandDI1FallingEdge, text list: 'CommandOnTerminalEvent'
        Textfield (15,175 170x30), "DI2 rising edge"
        ComboBoxInteger (205,175 250x30), variable: Communication.eCommandDI2RisingEdge, text list: 'CommandOnTerminalEvent'
        Textfield (15,225 170x30), "DI2 falling edge"
        ComboBoxInteger (205,225 250x30), variable: Communication.eCommandDI2FallingEdge, text list: 'CommandOnTerminalEvent'
        Button (220,330 200x40), "Write parameters"
            OnMouseClick: execute { Communication.bInitialize := TRUE; }
        Button (10,330 200x40), "Write default values"
            OnMouseClick: execute { Communication.bDefaultValues := TRUE; }
        Button (10,388 260x40), "Reset inactive process image"
            OnMouseClick: execute { Communication.bResetInactiveProcessImage := TRUE; }
        Checkbox (15,275 35x30), variable: Communication.bDoNotLockProcessImage
        Textfield (50,267 340x45), "Do not lock process image in case of DALI commands from DI1 or DI2"
    Image (481,135 316x300), image: ImagePool.KL6821
    Group (350,10 330x30)
        Checkbox (0,0 34x30), variable: Communication.bInternalPowerSupplyDisabled
        Textfield (30,0 294x30), "Internal DALI power supply disabled"
    Group (10,5 170x40)
        Textfield (0,0 110x40), "DALI Line:"
        Button (90,0 80x40), "%d", text variable: GVL_Internal.nDALILine
            OnMouseClick: write the text variable via Default, min 1, max 10, title "Choose line"
END_VISUALIZATION

// ---- VISUs/Visu_DALICommissioning/Visu_Part102Commands.TcVIS
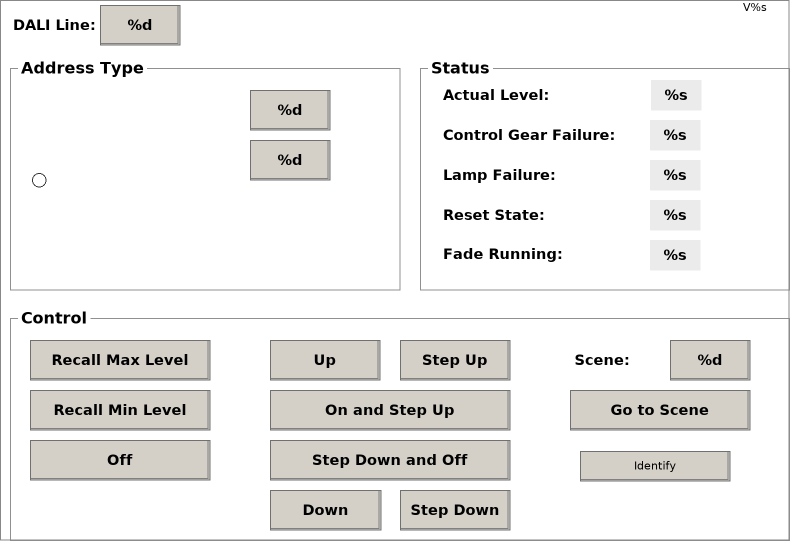
VISUALIZATION Visu_Part102Commands  // 790x541
    GroupBox (10,310 780x231), "Control"
        Button (20,130 180x40), "Off"
            OnMouseClick: execute { DALI_Commissioning.fbPart102Commands.bOff := TRUE; }
        Button (20,80 180x40), "Recall Min Level"
            OnMouseClick: execute { DALI_Commissioning.fbPart102Commands.bRecallMinLevel := TRUE; }
        Button (20,30 180x40), "Recall Max Level"
            OnMouseClick: execute { DALI_Commissioning.fbPart102Commands.bRecallMaxLevel := TRUE; }
        Button (260,180 111x40), "Down"
            OnMouseClick: execute { DALI_Commissioning.fbPart102Commands.bDown := TRUE; }
        Button (390,180 110x40), "Step Down"
            OnMouseClick: execute { DALI_Commissioning.fbPart102Commands.bStepDown := TRUE; }
        Button (260,130 240x40), "Step Down and Off"
            OnMouseClick: execute { DALI_Commissioning.fbPart102Commands.bStepDownAndOff := TRUE; }
        Button (660,30 80x40), "%d", text variable: DALI_Commissioning.fbPart102Commands.nScene
            OnMouseClick: write the text variable via Default, min 0, max 15, title "Insert scene number"
        Textfield (550,35 85x30), "Scene:"
        Button (560,80 180x40), "Go to Scene"
            OnMouseClick: execute { DALI_Commissioning.fbPart102Commands.bGotoScene := TRUE; }
        Button (260,80 240x40), "On and Step Up"
            OnMouseClick: execute { DALI_Commissioning.fbPart102Commands.bOnAndStepUp := TRUE; }
        Button (260,30 110x40), "Up"
            OnMouseClick: execute { DALI_Commissioning.fbPart102Commands.bUp := TRUE; }
        Button (390,30 110x40), "Step Up"
            OnMouseClick: execute { DALI_Commissioning.fbPart102Commands.bStepUp := TRUE; }
        Button (570,141 150x30), "Identify"
            OnMouseDown: execute { DALI_Commissioning.fbPart102Commands.bIdentify202 := TRUE; }
    GroupBox (420,60 370x230), "Status"
        Textfield (20,20 200x30), "Actual Level:"
        Textfield (20,60 200x30), "Control Gear Failure:"
        Textfield (231,20 50x30), "%s", text variable: DALI_Commissioning.fbPart102Commands.sActualLevel
        Textfield (230,60 50x30), "%s", text variable: DALI_Commissioning.fbPart102Commands.sControlGearFailure
        Textfield (20,100 200x30), "Lamp Failure:"
        Textfield (230,100 50x30), "%s", text variable: DALI_Commissioning.fbPart102Commands.sLampFailure
        Textfield (20,140 200x30), "Reset State:"
        Textfield (230,140 50x30), "%s", text variable: DALI_Commissioning.fbPart102Commands.sResetState
        Textfield (20,180 200x28), "Fade Running:"
        Textfield (230,180 50x30), "%s", text variable: DALI_Commissioning.fbPart102Commands.sFadeRunning
    GroupBox (10,60 390x230), "Address Type"
        Button (240,30 80x40), "%d", text variable: DALI_Commissioning.fbPart102Commands.nShortAddress
            OnMouseClick: write the text variable via Default, min 0, max 63, title "Insert Short Address"
            OnMouseClick: execute {  }
        RadioButton (20,20 190x200), variable: DALI_Commissioning.fbPart102Commands.eAddressType
            Areas[0]: Text=Short Address
            Areas[1]: Text=Group Address
            Areas[2]: Text=Broadcast
            Areas[3]: Text=Unaddressed
        Button (240,80 80x40), "%d", text variable: DALI_Commissioning.fbPart102Commands.nGroupAddress
            OnMouseClick: write the text variable via Default, min 0, max 15, title "Insert Group Address"
    Rectangle (720,0 70x15), "V%s", text variable: stLibVersion_Tc3_DALI_PLC_Commissioning_Tool.sVersion
    Group (10,5 170x40)
        Textfield (0,0 110x40), "DALI Line:"
        Button (90,0 80x40), "%d", text variable: GVL_Internal.nDALILine
            OnMouseClick: write the text variable via Default, min 1, max 10, title "Choose line"
END_VISUALIZATION

// ---- VISUs/Visu_DALICommissioning/Visu_Part102MemoryBank.TcVIS
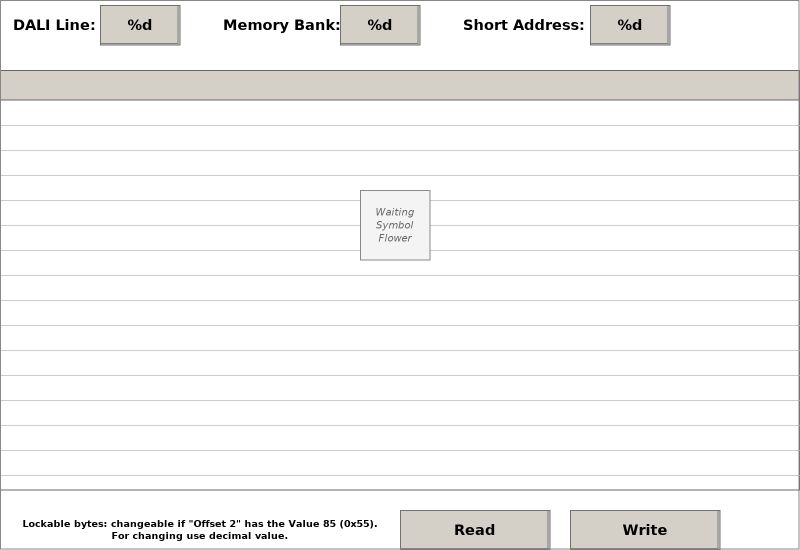
VISUALIZATION Visu_Part102MemoryBank  // 800x550
    Table (0,70 800x420), data array: DALI_Commissioning.fbPart102MemoryPages.aMemoryBank
        p1137915858: DALI_Commissioning.fbPart102MemoryPages.nOffset
        p3854506369: DALI_Commissioning.fbPart102MemoryPages.aMemoryBank[INDEX].sOffset
        p1892666644: DALI_Commissioning.fbPart102MemoryPages.aMemoryBank[INDEX].sName
        p338671338: DALI_Commissioning.fbPart102MemoryPages.aMemoryBank[INDEX].nValueDec
        p2170511999: DALI_Commissioning.fbPart102MemoryPages.aMemoryBank[INDEX].nValueHex
        p1755163831: Value Dec
        p4092479075: Value Hex
        Columns.Column.[2].Template: DALI_Commissioning.fbPart102MemoryPages.aNoValue[INDEX]; OnMouseClick: write the text variable via Default, min 0, max 255, title "Lockable variable decimal"
        Columns.Column.[0].Template: DALI_Commissioning.fbPart102MemoryPages.aNoValue[INDEX]
        Columns.Column.[1].Template: DALI_Commissioning.fbPart102MemoryPages.aNoValue[INDEX]
        Columns.Column.[3].Template: DALI_Commissioning.fbPart102MemoryPages.aNoValue[INDEX]; OnMouseClick: write the text variable via Default, title "Lockable variable hexadecimal"
    Button (400,510 150x40), "Read"
        OnMouseClick: execute { DALI_Commissioning.fbPart102MemoryPages.bRead := TRUE; }
    Button (570,510 150x40), "Write"
        OnMouseClick: execute { DALI_Commissioning.fbPart102MemoryPages.bWrite := TRUE; }
    Textfield (15,510 370x40), "Lockable bytes: changeable if "Offset 2" has the Value 85 (0x55). For changing use decimal value."
    WaitingSymbolFlower (360,190 70x70), invisible if: DALI_Commissioning.fbPart102MemoryPages.bHideWaitSymbol
    Textfield (460,5 130x40), "Short Address:"
    Button (590,5 80x40), "%d", text variable: DALI_Commissioning.fbPart102MemoryPages.nAddress
        OnMouseClick: write the text variable via Default, min 0, max 63, title "Insert Short Address"
    Textfield (220,5 120x40), "Memory Bank:"
    Button (340,5 80x40), "%d", text variable: DALI_Commissioning.fbPart102MemoryPages.nMemoryBank
        OnMouseClick: write the text variable via Default, min 0, max 255, title "Insert Memory Bank"
    Group (10,5 170x40)
        Textfield (0,0 110x40), "DALI Line:"
        Button (90,0 80x40), "%d", text variable: GVL_Internal.nDALILine
            OnMouseClick: write the text variable via Default, min 1, max 10, title "Choose line"
END_VISUALIZATION

// ---- VISUs/Visu_DALICommissioning/Visu_Part103Addressing.TcVIS
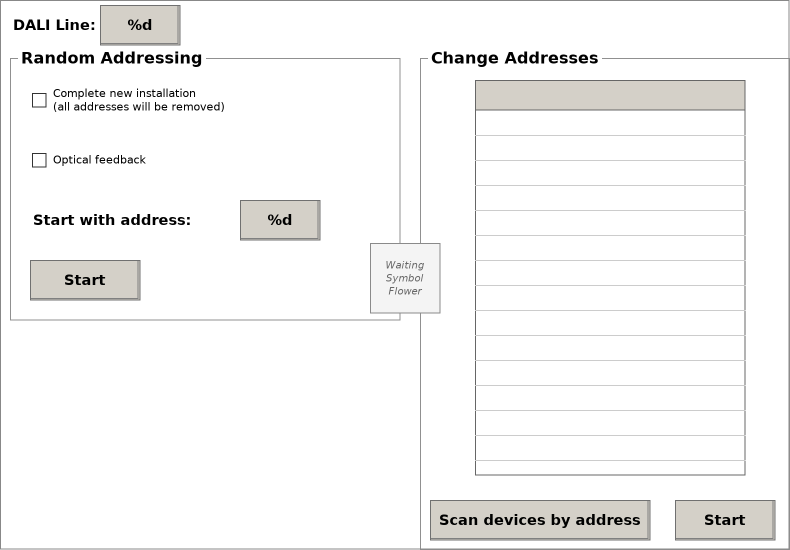
VISUALIZATION Visu_Part103Addressing  // 790x550
    GroupBox (420,50 370x500), "Change Addresses"
        Table (55,30 270x395), data array: DALI_Commissioning.fbPart103Addressing.aChangeAddressList
            p3854506369: DALI_Commissioning.fbPart103Addressing.aChangeAddressList[INDEX].nOldAddress
            p1892666644: DALI_Commissioning.fbPart103Addressing.aChangeAddressList[INDEX].nNewAddress
            p338671338: DALI_Commissioning.fbPart103Addressing.aChangeAddressList[INDEX].nRandomAddress
            p2170511999: DALI_Commissioning.fbPart103Addressing.aChangeAddressList[INDEX].nErrors
            Columns.Column.[0].Template: DALI_Commissioning.fbPart103Addressing.aNoShortAddress[INDEX]
            Columns.Column.[1].Template: DALI_Commissioning.fbPart103Addressing.aNoShortAddress[INDEX]; OnMouseClick: write the text variable via Default, min 0, max 63, title "New Short Address"
        Button (255,450 100x40), "Start"
            OnMouseClick: execute { DALI_Commissioning.fbPart103Addressing.bStartChangeAddress := TRUE; }
        Button (10,450 220x40), "Scan devices by address"
            OnMouseClick: execute { DALI_Commissioning.fbPart103Addressing.bScanDevices := TRUE; }
    GroupBox (10,50 390x270), "Random Addressing"
        Button (20,210 110x40), "Start"
            OnMouseClick: execute { DALI_Commissioning.fbPart103Addressing.bStartRandomAddressing := TRUE; }
        Checkbox (20,30 360x40), "Complete new installation (all addresses will be removed)", variable: DALI_Commissioning.fbPart103Addressing.bNewInstallation
        Checkbox (20,90 360x40), "Optical feedback", variable: DALI_Commissioning.fbPart103Addressing.bOpticalFeedback
        Textfield (20,150 200x40), "Start with address:"
        Button (230,150 80x40), "%d", text variable: DALI_Commissioning.fbPart103Addressing.nStartAddress
            OnMouseClick: write DALI_Commissioning.fbPart103Addressing.nStartAddress via Default, min 0, max 63, title "Insert Short Address"
    WaitingSymbolFlower (370,243 70x70), invisible if: DALI_Commissioning.fbPart103Addressing.bHideWaitSymbol
    Group (10,5 170x40)
        Textfield (0,0 110x40), "DALI Line:"
        Button (90,0 80x40), "%d", text variable: GVL_Internal.nDALILine
            OnMouseClick: write the text variable via Default, min 1, max 10, title "Choose line"
END_VISUALIZATION

// ---- VISUs/Visu_DALICommissioning/Visu_Part103Parameters.TcVIS
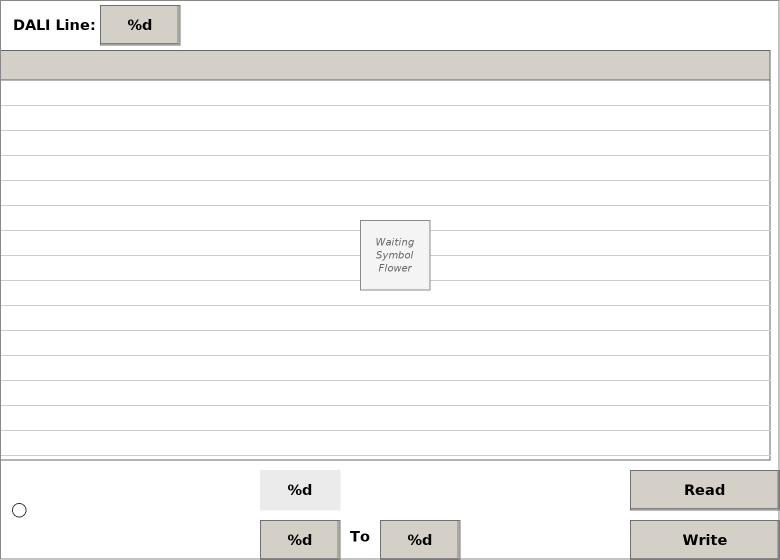
VISUALIZATION Visu_Part103Parameters  // 780x560
    Table (0,50 770x410), data array: DALI_Commissioning.fbPart103Parameters.aParameters
        p1137915858: DALI_Commissioning.fbPart103Parameters.nSelectedAddress
        p3854506369: DALI_Commissioning.fbPart103Parameters.aParameters[INDEX].nOperatingMode
        p1892666644: DALI_Commissioning.fbPart103Parameters.aParameters[INDEX].sInstanceType0
        p338671338: DALI_Commissioning.fbPart103Parameters.aParameters[INDEX].sInstanceType1
        p2170511999: DALI_Commissioning.fbPart103Parameters.aParameters[INDEX].sInstanceType2
        p3723444502: DALI_Commissioning.fbPart103Parameters.aParameters[INDEX].sInstanceType3
        p1218418051: DALI_Commissioning.fbPart103Parameters.aParameters[INDEX].sInstanceType4
        p511219082: IT0 (Generic Input)
        p1755163831: IT1 (PushButton)
        p4092479075: IT2 (Absolute Input)
        p2237128397: IT3 (Occupancy)
        p505689113: IT4 (Light Sensor)
        Columns.Column.[0].Template: OnMouseClick: write the text variable via Default, min 0, max 255, title "Insert Operating Mode 0, 128-255"
    RadioButton (10,460 230x100), variable: DALI_Commissioning.fbPart103Parameters.nAddressRange
        Areas[0]: Text=Single Short Address
        Areas[1]: Text=Short Address Range
    Textfield (260,470 80x40), "%d", text variable: DALI_Commissioning.fbPart103Parameters.nSelectedAddress
    Button (260,520 80x40), "%d", text variable: DALI_Commissioning.fbPart103Parameters.nStartAddress
        OnMouseClick: write the text variable via Default, min 0, max 63, title "Insert Short Address"
    Button (380,520 80x40), "%d", text variable: DALI_Commissioning.fbPart103Parameters.nEndAddress
        OnMouseClick: write the text variable via Default, min 0, max 63, title "Insert Short Address"
    Button (630,470 150x40), "Read"
        OnMouseClick: execute { DALI_Commissioning.fbPart103Parameters.bRead := true; }
    Button (630,520 150x40), "Write"
        OnMouseClick: execute { DALI_Commissioning.fbPart103Parameters.bWrite := true; }
    Textfield (335,521 50x31), "To"
    WaitingSymbolFlower (360,220 70x70), invisible if: DALI_Commissioning.fbPart103Parameters.bHideWaitSymbol
    Group (10,5 170x40)
        Textfield (0,0 110x40), "DALI Line:"
        Button (90,0 80x40), "%d", text variable: GVL_Internal.nDALILine
            OnMouseClick: write the text variable via Default, min 1, max 10, title "Choose line"
END_VISUALIZATION

// ---- VISUs/Visu_DALICommissioning/Visu_Part300GenericDevice.TcVIS
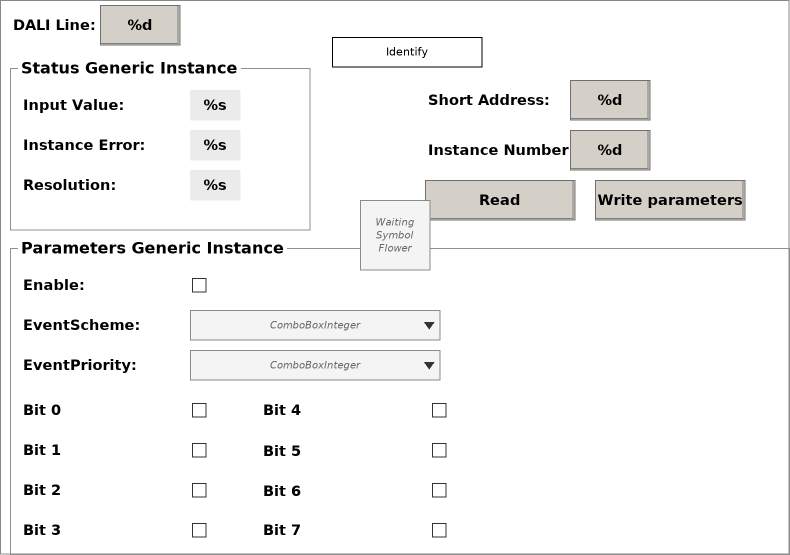
VISUALIZATION Visu_Part300GenericDevice  // 790x555
    GroupBox (10,240 780x315), "Parameters Generic Instance"
        Textfield (10,30 150x30), "Enable:"
        Checkbox (180,30 30x30), variable: DALI_Commissioning.fbPart300GenericDevice.bEnable
        Textfield (10,110 150x30), "EventPriority:"
        Textfield (10,195 100x30), "Bit 1"
        Textfield (10,155 100x30), "Bit 0"
        Checkbox (180,155 30x30), variable: DALI_Commissioning.fbPart300GenericDevice.bBit0
        Checkbox (180,195 30x30), variable: DALI_Commissioning.fbPart300GenericDevice.bBit1
        Textfield (10,235 100x30), "Bit 2"
        Textfield (250,155 100x30), "Bit 4"
        Textfield (250,196 100x30), "Bit 5"
        Checkbox (420,195 30x30), variable: DALI_Commissioning.fbPart300GenericDevice.bBit5
        Checkbox (420,155 30x30), variable: DALI_Commissioning.fbPart300GenericDevice.bBit4
        Checkbox (180,275 30x30), variable: DALI_Commissioning.fbPart300GenericDevice.bBit3
        Checkbox (180,235 30x30), variable: DALI_Commissioning.fbPart300GenericDevice.bBit2
        ComboBoxInteger (180,70 250x30), variable: DALI_Commissioning.fbPart300GenericDevice.eEventScheme, text list: 'EventScheme'
        Textfield (10,70 150x30), "EventScheme:"
        Textfield (250,236 100x30), "Bit 6"
        ComboBoxInteger (180,110 250x30), variable: DALI_Commissioning.fbPart300GenericDevice.eEventPriority, text list: 'EventPriority'
        Textfield (10,275 100x30), "Bit 3"
        Checkbox (420,235 30x30), variable: DALI_Commissioning.fbPart300GenericDevice.bBit6
        Checkbox (420,275 30x30), variable: DALI_Commissioning.fbPart300GenericDevice.bBit7
        Textfield (250,275 100x30), "Bit 7"
    GroupBox (10,60 300x170), "Status Generic Instance"
        Textfield (180,30 50x30), "%s", text variable: DALI_Commissioning.fbPart300GenericDevice.nInputValue
        Textfield (180,70 50x30), "%s", text variable: DALI_Commissioning.fbPart300GenericDevice.nInstanceError
        Textfield (180,110 50x30), "%s", text variable: DALI_Commissioning.fbPart300GenericDevice.nResolution
        Textfield (10,30 160x30), "Input Value:"
        Textfield (10,70 160x30), "Instance Error:"
        Textfield (10,110 160x30), "Resolution:"
    Button (425,180 150x40), "Read"
        OnMouseClick: execute { DALI_Commissioning.fbPart300GenericDevice.bRead := TRUE; }
    WaitingSymbolFlower (360,200 70x70), invisible if: DALI_Commissioning.fbPart300GenericDevice.bHideWaitSymbol
    Button (595,180 150x40), "Write parameters"
        OnMouseClick: execute { DALI_Commissioning.fbPart300GenericDevice.bWrite := TRUE; }
    Textfield (425,130 150x40), "Instance Number:"
    Textfield (425,80 150x40), "Short Address:"
    Button (570,80 80x40), "%d", text variable: DALI_Commissioning.fbPart300GenericDevice.nAddress
        OnMouseClick: write the text variable via Default, min 0, max 63, title "Insert Short Address"
    Button (570,130 80x40), "%d", text variable: DALI_Commissioning.fbPart300GenericDevice.nInstanceAddress
        OnMouseClick: write the text variable via Default, min 0, max 31, title "Insert instance number"
    Group (10,5 170x40)
        Textfield (0,0 110x40), "DALI Line:"
        Button (90,0 80x40), "%d", text variable: GVL_Internal.nDALILine
            OnMouseClick: write the text variable via Default, min 1, max 10, title "Choose line"
    Rectangle (332,37 150x30), "Identify"
        OnMouseDown: execute { DALI_Commissioning.fbPart300GenericDevice.bIdentify := TRUE; }
END_VISUALIZATION

// ---- VISUs/Visu_DALICommissioning/Visu_Part302AbsoluteInputDevice.TcVIS
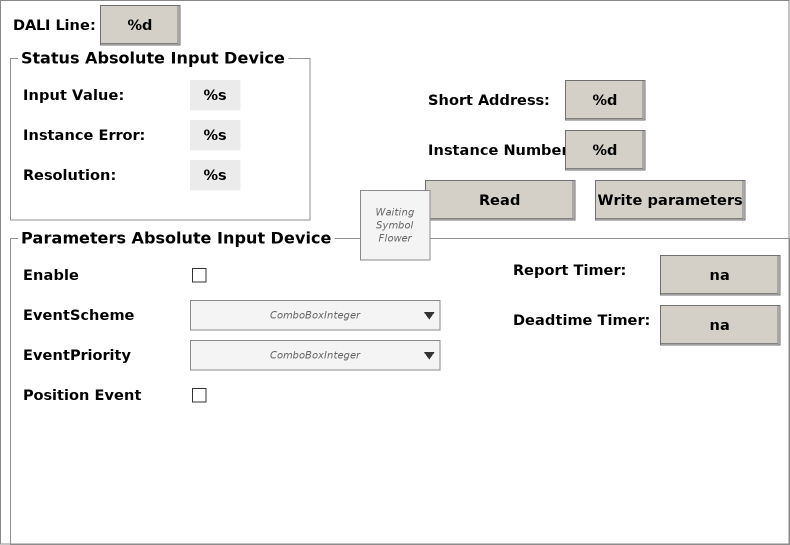
VISUALIZATION Visu_Part302AbsoluteInputDevice  // 790x545
    GroupBox (10,50 300x170), "Status Absolute Input Device"
        Textfield (10,30 160x30), "Input Value:"
        Textfield (10,70 160x30), "Instance Error:"
        Textfield (10,110 160x30), "Resolution:"
        Textfield (180,30 50x30), "%s", text variable: DALI_Commissioning.fbPart302AbsoluteInputDevice.nInputValue
        Textfield (180,70 50x30), "%s", text variable: DALI_Commissioning.fbPart302AbsoluteInputDevice.nInstanceError
        Textfield (180,110 50x30), "%s", text variable: DALI_Commissioning.fbPart302AbsoluteInputDevice.nResolution
    Button (425,180 150x40), "Read"
        OnMouseClick: execute { DALI_Commissioning.fbPart302AbsoluteInputDevice.bRead := TRUE; }
    GroupBox (10,230 780x315), "Parameters Absolute Input Device"
        Textfield (500,75 145x30), "Deadtime Timer:"
        Textfield (500,25 145x30), "Report Timer:"
        Textfield (10,30 150x30), "Enable"
        Button (650,25 120x40), "%d s", text variable: DALI_Commissioning.fbPart302AbsoluteInputDevice.nReport
            OnMouseClick: write DALI_Commissioning.fbPart302AbsoluteInputDevice.nReport via Default, min 0, max 255, title "Insert value for report timer"
        Button (650,75 120x40), "%d ms", text variable: DALI_Commissioning.fbPart302AbsoluteInputDevice.nDeadtime
            OnMouseClick: write DALI_Commissioning.fbPart302AbsoluteInputDevice.nDeadtime via Default, min 0, max 12750, title "Insert value for deadtime timer"
        Checkbox (180,30 30x30), variable: DALI_Commissioning.fbPart302AbsoluteInputDevice.bEnable
        Textfield (10,70 150x30), "EventScheme"
        ComboBoxInteger (180,70 250x30), variable: DALI_Commissioning.fbPart302AbsoluteInputDevice.eEventScheme, text list: 'EventScheme'
        Button (650,25 120x40), "na", invisible if: Not DALI_Commissioning.fbPart302AbsoluteInputDevice.bNoReportTimer, input disabled if: Not DALI_Commissioning.fbPart302AbsoluteInputDevice.bNoReportTimer
        Button (650,75 120x40), "na", invisible if: Not DALI_Commissioning.fbPart302AbsoluteInputDevice.bNoDeadtimeTimer, input disabled if: Not DALI_Commissioning.fbPart302AbsoluteInputDevice.bNoDeadtimeTimer
        Textfield (10,110 150x30), "EventPriority"
        Textfield (10,150 150x30), "Position Event"
        ComboBoxInteger (180,110 250x30), variable: DALI_Commissioning.fbPart302AbsoluteInputDevice.eEventPriority, text list: 'EventPriority'
        Checkbox (180,150 30x30), variable: DALI_Commissioning.fbPart302AbsoluteInputDevice.bPositionEventEnabled
    WaitingSymbolFlower (360,190 70x70), invisible if: DALI_Commissioning.fbPart302AbsoluteInputDevice.bHideWaitSymbol
    Button (595,180 150x40), "Write parameters"
        OnMouseClick: execute { DALI_Commissioning.fbPart302AbsoluteInputDevice.bWrite := TRUE; }
    Group (10,5 170x40)
        Textfield (0,0 110x40), "DALI Line:"
        Button (90,0 80x40), "%d", text variable: GVL_Internal.nDALILine
            OnMouseClick: write the text variable via Default, min 1, max 10, title "Choose line"
    Textfield (425,80 130x40), "Short Address:"
    Button (565,80 80x40), "%d", text variable: DALI_Commissioning.fbPart302AbsoluteInputDevice.nAddress
        OnMouseClick: write DALI_Commissioning.fbPart302AbsoluteInputDevice.nAddress via Default, min 0, max 63, title "Insert Short Address"
    Textfield (425,130 150x40), "Instance Number:"
    Button (565,130 80x40), "%d", text variable: DALI_Commissioning.fbPart302AbsoluteInputDevice.nInstanceAddress
        OnMouseClick: write DALI_Commissioning.fbPart302AbsoluteInputDevice.nInstanceAddress via Default, min 0, max 31, title "Insert instance number"
END_VISUALIZATION
